FUNCTION_BLOCK FB_UnixTimeStampGlobal
(*
    Runs FB_UnixTimeStamp and stuffs the result into this library's GVL
    2019-10-09 Zachary Lentz
*)
VAR_INPUT
    // If TRUE, we will update the output on this cycle.
    bExecute: BOOL;
END_VAR
VAR_OUTPUT
END_VAR
VAR
    fbTimeStamp: FB_UnixTimeStamp;
END_VAR

fbTimeStamp(
    bExecute := bExecute,
    fTime => DefaultGlobals.fTimeStamp);

END_FUNCTION_BLOCK

(* stored: Version 1.1.0.1
   POU FB_UnixTimeStampGlobal: Id {626742ce-ebb0-42d8-8b96-83167f2ea362}, SpecialFunc None *)
